(* PLC project Unnamed, Unknown Unnamed 1 *)
(* stored: creationDateTime 2024-03-06T12:20:15, modificationDateTime 2024-03-08T10:29:22 *)

TYPE S_FA_STATUS : STRUCT
  BART_Hand : BOOL := true;
  BART_Auto : BOOL := false;
  Stoerung : BOOL := false;
  Stoer_Quit : BOOL := false;
  NotHalt : BOOL := false;
  Takt : BOOL := false;
END_STRUCT;
END_TYPE

(* Aktor 5/2 Magnetventil *)
FUNCTION_BLOCK AKT_5_2_MV
  VAR_INPUT
    status : S_FA_STATUS;  (* P1 soll angefahren werden (Feder forsiert P1) *)
    Hand_P1 : BOOL;  (* P1 soll angefahren werden (Feder forsiert P1) *)
    Hand_P2 : BOOL;  (* P2 soll angefahren werden (Feder arbeitet gegen P2) *)
  END_VAR
  VAR
    SR0 : SR;
  END_VAR
  VAR_OUTPUT
    s_MV_P2_FF : BOOL;  (* Ausgabe um das Signal -1Y2 ansteuern zu können *)
  END_VAR
  VAR
    DebugBoolean : BOOL;
    TON0 : TON;
  END_VAR
  VAR CONSTANT
    const_T_Laufzeit_P2 : TIME := T#10s;
  END_VAR
  VAR_INPUT
    SEN_P1 : BOOL;  (* Sensor Position 1 activates, the cylinder has made it to P1 *)
    SEN_P2 : BOOL;  (* Sensor Position 2 activates, the cylinder has made it to P2 *)
  END_VAR

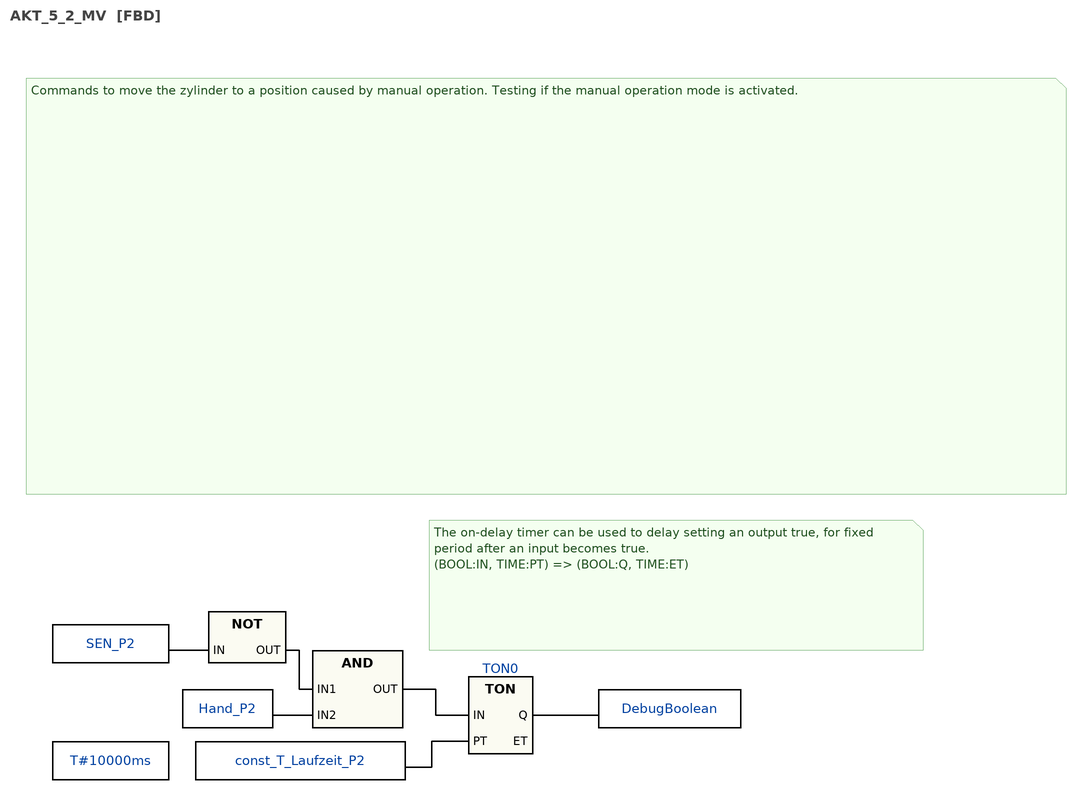
(* FBD diagram, written out as Structured Text *)
(* Commands to move the zylinder to a position caused by manual operation. Testing if the manual operation mode is activated. *)
SR0(S1 := status.BART_Hand AND Hand_P2, R := status.BART_Hand AND Hand_P1);
s_MV_P2_FF := SR0.Q1;
(* The on-delay timer can be used to delay setting an output true, for fixed period after an input becomes true.
 (BOOL:IN, TIME:PT) => (BOOL:Q, TIME:ET) *)
TON0(IN := NOT SEN_P2 AND Hand_P2, PT := const_T_Laufzeit_P2);
DebugBoolean := TON0.Q;
(* drawn but not wired to any output: T#10000ms *)
END_FUNCTION_BLOCK

FUNCTION FA_SERV : BOOL
  VAR_INPUT
    status : S_FA_STATUS;
    BART_Hand : BOOL;
    BART_Auto : BOOL;
    Stoerung : BOOL;
    Stoer_Quit : BOOL;
    NotHalt : BOOL;
  END_VAR

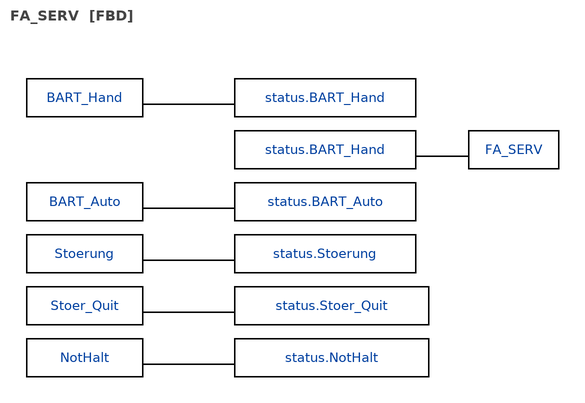
(* FBD diagram, written out as Structured Text *)
status.BART_Hand := BART_Hand;
FA_SERV := status.BART_Hand;
status.BART_Auto := BART_Auto;
status.Stoerung := Stoerung;
status.Stoer_Quit := Stoer_Quit;
status.NotHalt := NotHalt;
END_FUNCTION

PROGRAM program0_POU
  VAR
    FA_Start_T_HMI : BOOL;  (* Defined in the Res0 resource *)
    FA_Init_T_HMI : BOOL;  (* Defined in the Res0 resource *)
    FA_Sonder_T_HMI : BOOL;  (* Defined in the Res0 resource *)
    FA_Stop_T_HMI : BOOL;  (* Defined in the Res0 resource *)
    FA_BART_Hand_T_HMI : BOOL := true;  (* Defined in the Res0 resource *)
    FA_BART_Auto_T_HMI : BOOL;  (* Defined in the Res0 resource *)
    FA_BART_Auto_Einzel_T_HMI : BOOL;  (* Defined in the Res0 resource *)
    FA_Stoerung_T_HMI : BOOL;  (* Defined in the Res0 resource *)
    FA_Stoer_Quit_T_HMI : BOOL;  (* Defined in the Res0 resource *)
    FA_NotHalt_T_HMI : BOOL;  (* Defined in the Res0 resource *)
    DebugBoolean : BOOL;  (* Defined in the Res0 resource *)
  END_VAR
  VAR_EXTERNAL
    global_status : S_FA_STATUS;  (* Defined in the Res0 resource *)
  END_VAR
  VAR
    AKT_5_2_MV0 : AKT_5_2_MV;
    Zyl1_T_P1_HMI : BOOL;
    Zyl1_T_P2_HMI : BOOL;
    s_MV_P2_FF : BOOL;  (* -1Y2 Zylinder 1, Magnetventil Spule *)
    SEN_P1_T_HMI : BOOL := true;
    SEN_P2_T_HMI : BOOL := false;
  END_VAR

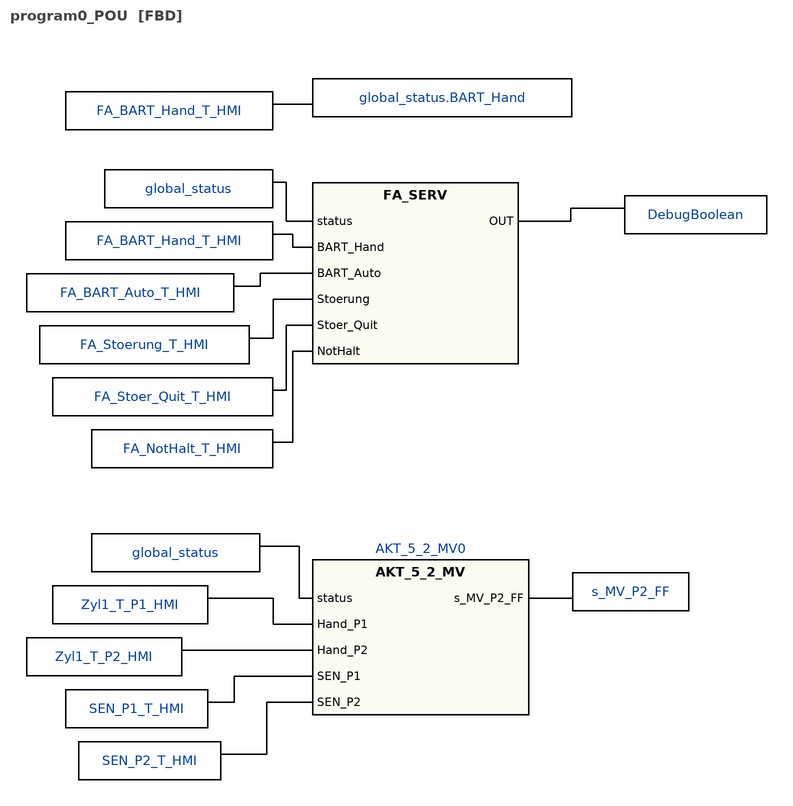
(* FBD diagram, written out as Structured Text *)
global_status.BART_Hand := FA_BART_Hand_T_HMI;
DebugBoolean := FA_SERV(global_status, FA_BART_Hand_T_HMI, FA_BART_Auto_T_HMI, FA_Stoerung_T_HMI, FA_Stoer_Quit_T_HMI, FA_NotHalt_T_HMI);
AKT_5_2_MV0(status := global_status, Hand_P1 := Zyl1_T_P1_HMI, Hand_P2 := Zyl1_T_P2_HMI, SEN_P1 := SEN_P1_T_HMI, SEN_P2 := SEN_P2_T_HMI);
s_MV_P2_FF := AKT_5_2_MV0.s_MV_P2_FF;
END_PROGRAM

FUNCTION_BLOCK FA
  VAR
    Status : S_FA_STATUS;
  END_VAR

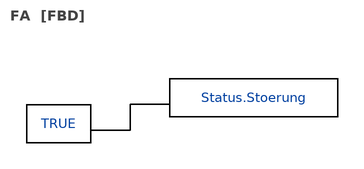
(* FBD diagram, written out as Structured Text *)
Status.Stoerung := TRUE;
END_FUNCTION_BLOCK

CONFIGURATION Config0
  RESOURCE Res0 ON PLC
    VAR_GLOBAL
      global_status : S_FA_STATUS;
    END_VAR
    TASK task0(INTERVAL := T#20ms, PRIORITY := 0);
    PROGRAM instance0 WITH task0 : program0_POU;
  END_RESOURCE
END_CONFIGURATION
